Staubli VAL3: onEdit.pgx

public program onEdit(string& x_sItem[])
  local string l_sPath
  local string l_sName
  local num l_nResult
begin
  // DEFINE YOUR ITEM
  call getTrajType(saveData:sTrajTypeUsing)
  // load the trajectory
  call load(x_sItem,l_nResult)
  if size(x_sItem)>1
    // give back the path
    l_sPath="Disk://trajectory/page_viewTraj"
    x_sItem[1]=x_sItem
    x_sItem=l_sPath
    // init
    tAppro={0,0,0,0,0,0}
    tPointTo={0,0,0,0,0,0}
    nZeta=0
  endIf
end
